// TwinCAT 3 PLC project TcPLCopenOopExample
// ProgramVersion: 3.1.4023.0
// libraries:
//   Tc2_Standard, * (Beckhoff Automation GmbH)
//   Tc2_System, * (Beckhoff Automation GmbH)
//   Tc3_Module, * (Beckhoff Automation GmbH)
// project tree:
//   DUTs/ stCBMLInfo.TcDUT
//   / PlcTask.TcTTO
//   POUs/ FB_Boiler.TcPOU, FB_Drum.TcPOU, FB_ErrorHandler.TcPOU, ITF_Device.TcIO, ITF_ErrorHandlerSubject.TcIO, MAIN.TcPOU
// real-time tasks:
//   TASK PlcTask: cycle T#10ms, priority 20, ADS port 350

CONFIGURATION TcPLCopenOopExample
    RESOURCE PLC ON TwinCAT3
        TASK PlcTask(INTERVAL := T#10ms, PRIORITY := 20);
        PROGRAM MAIN WITH PlcTask : MAIN;
    END_RESOURCE
END_CONFIGURATION

// ---- DUTs/stCBMLInfo.TcDUT
TYPE stCBMLInfo :
STRUCT
	sName		: STRING;
	xError 		: BOOL;
	iErrorID 	: INT;
END_STRUCT
END_TYPE

// ---- POUs/ITF_Device.TcIO
INTERFACE ITF_Device

METHOD M_GetState : BOOL
VAR_OUTPUT
	O_stCBMLInfo : stCBMLInfo;
END_VAR
END_METHOD

METHOD M_SetName : BOOL
VAR_INPUT
	sName		: STRING;
END_VAR
END_METHOD

PROPERTY P_stCBMLInfo : stCBMLInfo
GET
END_GET
SET
END_SET
END_PROPERTY

END_INTERFACE

// ---- POUs/ITF_ErrorHandlerSubject.TcIO
INTERFACE ITF_ErrorHandlerSubject

METHOD AttachDevice : BOOL
VAR_INPUT
	itfDevice 	: ITF_Device;
END_VAR
END_METHOD

END_INTERFACE

// ---- POUs/MAIN.TcPOU
PROGRAM MAIN
VAR
	fbErrorHandler: FB_ErrorHandler;
	fbBoiler1: FB_Boiler;
	fbBoiler2: FB_Boiler;
END_VAR


fbBoiler1(itfErrorHandler:=fbErrorHandler );
fbBoiler2(itfErrorHandler:=fbErrorHandler );

fbErrorHandler();

END_PROGRAM

// ---- POUs/FB_ErrorHandler.TcPOU
FUNCTION_BLOCK FB_ErrorHandler IMPLEMENTS ITF_ErrorHandlerSubject
VAR_INPUT
END_VAR
VAR_OUTPUT
END_VAR
VAR
	_arStCBMLInfo		: ARRAY [0..100] OF stCBMLInfo;
	arItfDeviceObserver : ARRAY [0..100] OF ITF_Device;
	uiFc				: UINT;
END_VAR

FOR uiFc:=0 TO 100 BY 1 DO
	IF (arItfDeviceObserver[uiFc] <> 0) THEN
		_arStCBMLInfo[uiFc]:= arItfDeviceObserver[uiFc].P_stCBMLInfo;
	END_IF
END_FOR

METHOD AttachDevice : BOOL
VAR_INPUT
	itfDevice 	: ITF_Device;
END_VAR

VAR 
	uiFc 		: UINT;
END_VAR
FOR uiFc:= 0 TO 100 BY 1 DO
	IF (itfDevice <> 0) AND (arItfDeviceObserver[uiFc] = 0) THEN
		arItfDeviceObserver[uiFc] := itfDevice;
		EXIT;
	END_IF
END_FOR
END_METHOD

END_FUNCTION_BLOCK

// ---- POUs/FB_Boiler.TcPOU
FUNCTION_BLOCK FB_Boiler 
VAR_INPUT
	itfErrorHandler		: ITF_ErrorHandlerSubject;
END_VAR
VAR_OUTPUT
END_VAR
VAR
	xInit				: BOOL;
	fbDrum1				: FB_Drum;
	fbDrum2				: FB_Drum;
END_VAR

IF (NOT xInit) THEN
	xInit := TRUE;
	fbDrum1.M_SetName('Drum1');
	fbDrum2.M_SetName('Drum2');
	
	
	IF (itfErrorHandler <> 0) THEN
		itfErrorHandler.AttachDevice(fbDrum1);
		itfErrorHandler.AttachDevice(fbDrum2);
	END_IF
END_IF

END_FUNCTION_BLOCK

// ---- POUs/FB_Drum.TcPOU
FUNCTION_BLOCK FB_Drum IMPLEMENTS  ITF_Device
VAR_INPUT
END_VAR
VAR_OUTPUT
END_VAR
VAR
	_stCBMLInfo 	: stCBMLInfo;
END_VAR

{warning 'add method implementation '}
METHOD M_GetState : BOOL;

VAR_OUTPUT
	O_stCBMLInfo : stCBMLInfo;
END_VAR
O_stCBMLInfo := _stCBMLInfo;
END_METHOD

{warning 'add method implementation '}
METHOD M_SetName : BOOL
VAR_INPUT
	sName	: STRING;
END_VAR
_stCBMLInfo.sName := sName;
END_METHOD

{warning 'add property implementation'}
PROPERTY P_stCBMLInfo : stCBMLInfo
GET
P_stCBMLInfo := _stCBMLInfo;
END_GET
SET
END_SET
END_PROPERTY

END_FUNCTION_BLOCK
